// TIA Portal V20 export
FUNCTION_BLOCK "COLLECTIVE_OR_SIGNAL_FB"   // FB41, LAD
TITLE = COLLECTIVE_OR_SIGNAL_FB / COLLECTIVE_OR_SIGNAL_FC
{ S7_Optimized_Access := 'TRUE' }
AUTHOR : Tesla
FAMILY : Alarm_PD
VERSION : 1.0
// Der Baustein verodert 16 Eingangssignale (SIGNAL_1…SIGNAL_16) zu einem Ausgangssignal (COLLECTIVE_SIGNAL).
// Verwendungszweck (Beispiel): Zur Bildung eines Sammelsignals (z.B. für eine Sammelfehler-Leuchte für "Alarme", "Warnungen", "Infos") aus den Kategorie-Informationen der ProDiag-IDBs.
// The block converts 16 input signals (SIGNAL_1 ... SIGNAL_16) into an output signal (COLLECTIVE_SIGNAL), with OR-function.
// Purpose (example): To form a collection signal (e.g., a collective error light for "alarms," "warnings," "info") from the category information of the ProDiag IDBs.
// block converts 16 输入 信号 (SIGNAL_1 ... SIGNAL_16) into an 输出 信号 (COLLECTIVE_SIGNAL), 有 或者-功能.
// Purpose (例子): 到 form a collection 信号 (e.g., a collective 错误 light 给 "警报," "warnings," "信息") 从  类别 信息 of  ProDiag IDBs.
// stored: MemoryReserve 100, SetENOAutomatically false
   VAR_INPUT
      SIGNAL_1 { ExternalAccessible := 'False'; ExternalVisible := 'False'; ExternalWritable := 'False'} : Bool;   // Eingangs-Signal (Bool) / Input signal (Bool) / 输入 信号 (Bool)
      SIGNAL_2 { ExternalAccessible := 'False'; ExternalVisible := 'False'; ExternalWritable := 'False'} : Bool;   // Eingangs-Signal (Bool) / Input signal (Bool) / 输入 信号 (Bool)
      SIGNAL_3 { ExternalAccessible := 'False'; ExternalVisible := 'False'; ExternalWritable := 'False'} : Bool;   // Eingangs-Signal (Bool) / Input signal (Bool) / 输入 信号 (Bool)
      SIGNAL_4 { ExternalAccessible := 'False'; ExternalVisible := 'False'; ExternalWritable := 'False'} : Bool;   // Eingangs-Signal (Bool) / Input signal (Bool) / 输入 信号 (Bool)
      SIGNAL_5 { ExternalAccessible := 'False'; ExternalVisible := 'False'; ExternalWritable := 'False'} : Bool;   // Eingangs-Signal (Bool) / Input signal (Bool) / 输入 信号 (Bool)
      SIGNAL_6 { ExternalAccessible := 'False'; ExternalVisible := 'False'; ExternalWritable := 'False'} : Bool;   // Eingangs-Signal (Bool) / Input signal (Bool) / 输入 信号 (Bool)
      SIGNAL_7 { ExternalAccessible := 'False'; ExternalVisible := 'False'; ExternalWritable := 'False'} : Bool;   // Eingangs-Signal (Bool) / Input signal (Bool) / 输入 信号 (Bool)
      SIGNAL_8 { ExternalAccessible := 'False'; ExternalVisible := 'False'; ExternalWritable := 'False'} : Bool;   // Eingangs-Signal (Bool) / Input signal (Bool) / 输入 信号 (Bool)
      SIGNAL_9 { ExternalAccessible := 'False'; ExternalVisible := 'False'; ExternalWritable := 'False'} : Bool;   // Eingangs-Signal (Bool) / Input signal (Bool) / 输入 信号 (Bool)
      SIGNAL_10 { ExternalAccessible := 'False'; ExternalVisible := 'False'; ExternalWritable := 'False'} : Bool;   // Eingangs-Signal (Bool) / Input signal (Bool) / 输入 信号 (Bool)
      SIGNAL_11 { ExternalAccessible := 'False'; ExternalVisible := 'False'; ExternalWritable := 'False'} : Bool;   // Eingangs-Signal (Bool) / Input signal (Bool) / 输入 信号 (Bool)
      SIGNAL_12 { ExternalAccessible := 'False'; ExternalVisible := 'False'; ExternalWritable := 'False'} : Bool;   // Eingangs-Signal (Bool) / Input signal (Bool) / 输入 信号 (Bool)
      SIGNAL_13 { ExternalAccessible := 'False'; ExternalVisible := 'False'; ExternalWritable := 'False'} : Bool;   // Eingangs-Signal (Bool) / Input signal (Bool) / 输入 信号 (Bool)
      SIGNAL_14 { ExternalAccessible := 'False'; ExternalVisible := 'False'; ExternalWritable := 'False'} : Bool;   // Eingangs-Signal (Bool) / Input signal (Bool) / 输入 信号 (Bool)
      SIGNAL_15 { ExternalAccessible := 'False'; ExternalVisible := 'False'; ExternalWritable := 'False'} : Bool;   // Eingangs-Signal (Bool) / Input signal (Bool) / 输入 信号 (Bool)
      SIGNAL_16 { ExternalAccessible := 'False'; ExternalVisible := 'False'; ExternalWritable := 'False'} : Bool;   // Eingangs-Signal (Bool) / Input signal (Bool) / 输入 信号 (Bool)
   END_VAR
   VAR_OUTPUT
      COLLECTIVE_SIGNAL : Bool;   // Ausgangs-Summensignal (Bool) / Output Collective signal (Bool) / 输出 Collective 信号 (Bool)
   END_VAR
BEGIN

REGION Network 1: Ausgangs-Summensignal (Bool) / Output Collective signal (Bool) / 输出 Collective 信号 (Bool)
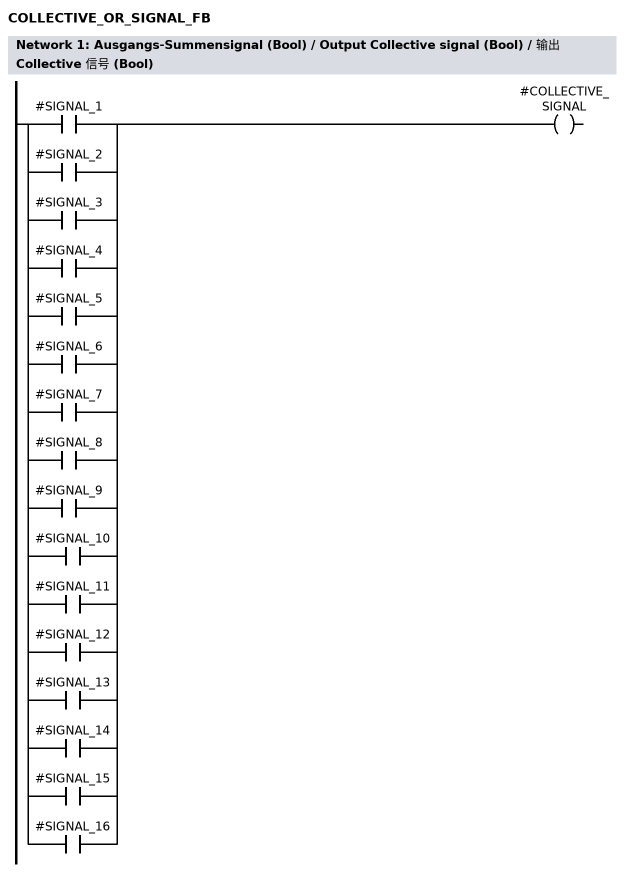
   RUNG wire#powerrail
      Contact( #SIGNAL_1 )
      wire#w1
      Coil( #COLLECTIVE_SIGNAL )
   END_RUNG
   RUNG wire#powerrail
      Contact( #SIGNAL_2 )
   END_RUNG wire#w1
   RUNG wire#powerrail
      Contact( #SIGNAL_3 )
   END_RUNG wire#w1
   RUNG wire#powerrail
      Contact( #SIGNAL_4 )
   END_RUNG wire#w1
   RUNG wire#powerrail
      Contact( #SIGNAL_5 )
   END_RUNG wire#w1
   RUNG wire#powerrail
      Contact( #SIGNAL_6 )
   END_RUNG wire#w1
   RUNG wire#powerrail
      Contact( #SIGNAL_7 )
   END_RUNG wire#w1
   RUNG wire#powerrail
      Contact( #SIGNAL_8 )
   END_RUNG wire#w1
   RUNG wire#powerrail
      Contact( #SIGNAL_9 )
   END_RUNG wire#w1
   RUNG wire#powerrail
      Contact( #SIGNAL_10 )
   END_RUNG wire#w1
   RUNG wire#powerrail
      Contact( #SIGNAL_11 )
   END_RUNG wire#w1
   RUNG wire#powerrail
      Contact( #SIGNAL_12 )
   END_RUNG wire#w1
   RUNG wire#powerrail
      Contact( #SIGNAL_13 )
   END_RUNG wire#w1
   RUNG wire#powerrail
      Contact( #SIGNAL_14 )
   END_RUNG wire#w1
   RUNG wire#powerrail
      Contact( #SIGNAL_15 )
   END_RUNG wire#w1
   RUNG wire#powerrail
      Contact( #SIGNAL_16 )
   END_RUNG wire#w1
   // the same network as SCL:
   #COLLECTIVE_SIGNAL := #SIGNAL_1 OR #SIGNAL_2 OR #SIGNAL_3 OR #SIGNAL_4 OR #SIGNAL_5 OR #SIGNAL_6 OR #SIGNAL_7 OR #SIGNAL_8 OR #SIGNAL_9 OR #SIGNAL_10 OR #SIGNAL_11 OR #SIGNAL_12 OR #SIGNAL_13 OR #SIGNAL_14 OR #SIGNAL_15 OR #SIGNAL_16;
END_REGION

NETWORK
TITLE = Baustein-Ende / End of block / 结束 of block
// ENO immer "1" setzen mit SET & SAVE / ENO always set to "1" with SET & SAVE / ENO 总是 设置 到 "1" 有 设置 & 保存
      SET;
      SAVE;
END_FUNCTION_BLOCK
